TYPE TermChannel :
STRUCT
	Status: WORD; (*бит XX.0 Underrange; бит ХХ.1 -Overrange; бит ХХ.6 - ERROR*)
	Value: INT;
END_STRUCT
END_TYPE

(* stored: Version 1.1.0.1, ProductVersion 3.1.4022.10
   DUT TermChannel: Id {17ebf9d7-4df1-4a5c-b266-a83ec78518bd} *)
